Fanuc KAREL source: kt00906.KL

-- PROVISIONAL review KL for V770-1; original PC SHA256 8b01f3c64c34e52295bdc9499560a9dd78482a8c40355bde74706f3f12f3eb2c
-- Incomplete behavior may be omitted. Consult companion uncertainty JSON. Do not deploy.
PROGRAM KT00906
%NOLOCKGROUP
BEGIN
  -- UNRESOLVED_PC offsets 5-31; opcodes 27,27,49,7E,AD,31,4A
  -- UNRESOLVED_PC offsets 36-40; opcodes 7F
END KT00906
